(* PLC project Unnamed, Unknown Unnamed 1 *)
(* stored: creationDateTime 2023-03-25T12:40:06, modificationDateTime 2023-03-28T19:18:31 *)

PROGRAM PPXYZ
  VAR
    START AT %IX100.0 : BOOL;
    STOP AT %IX100.1 : BOOL;
    SEN1 AT %IX100.2 : BOOL;
    SEN2 AT %IX100.3 : BOOL;
    CON1 AT %QX100.0 : BOOL;
    CON2 AT %QX100.1 : BOOL;
    GRAP AT %QX100.2 : BOOL;
    X AT %IW100 : INT;
    SPX AT %QW100 : INT;
    SPY AT %QW101 : INT;
    SPZ AT %QW102 : INT;
    DIGRED AT %QW103 : INT;
    VIR1 AT %QX0.0 : BOOL;
    VIR2 AT %QX0.1 : BOOL;
    VIR3 AT %QX0.2 : BOOL;
    VIR4 AT %QX0.3 : BOOL;
    VIR5 AT %QX0.4 : BOOL;
    VIR6 AT %QX0.5 : BOOL;
    VIR7 AT %QX0.6 : BOOL;
    VIR8 AT %QX0.7 : BOOL;
    Block1 AT %QX1.0 : BOOL;
    Block2 AT %QX1.1 : BOOL;
    Block3 AT %QX1.2 : BOOL;
    Block4 AT %QX1.3 : BOOL;
    GRABVIR1 AT %QX2.1 : BOOL;
    GRABVIR2 AT %QX2.2 : BOOL;
    GRABVIR3 AT %QX2.3 : BOOL;
    GRABVIR4 AT %QX2.4 : BOOL;
  END_VAR
  VAR
    TON0 : TON;
    TON1 : TON;
    TON2 : TON;
    TON3 : TON;
    TON4 : TON;
    TON5 : TON;
    TON6 : TON;
    TON7 : TON;
    TON8 : TON;
    TON9 : TON;
    TON10 : TON;
    TON11 : TON;
    TON12 : TON;
    TON13 : TON;
    TON14 : TON;
    TON15 : TON;
    TON16 : TON;
    TON17 : TON;
    TON18 : TON;
    TON19 : TON;
  END_VAR
  VAR  (* added by the conversion: wires and edge detectors of the diagram *)
    _MOVE77_ENO : BOOL;
    _MOVE77_OUT : INT;
    _MOVE8_ENO : BOOL;
    _MOVE8_OUT : INT;
    _MOVE12_ENO : BOOL;
    _MOVE12_OUT : INT;
    _MOVE16_ENO : BOOL;
    _MOVE16_OUT : INT;
    _MOVE20_ENO : BOOL;
    _MOVE20_OUT : INT;
    _MOVE29_ENO : BOOL;
    _MOVE29_OUT : INT;
    _MOVE69_ENO : BOOL;
    _MOVE69_OUT : INT;
    _MOVE40_ENO : BOOL;
    _MOVE40_OUT : INT;
    _MOVE44_ENO : BOOL;
    _MOVE44_OUT : INT;
    _MOVE48_ENO : BOOL;
    _MOVE48_OUT : INT;
    _MOVE52_ENO : BOOL;
    _MOVE52_OUT : INT;
    _MOVE61_ENO : BOOL;
    _MOVE61_OUT : INT;
    _MOVE139_ENO : BOOL;
    _MOVE139_OUT : INT;
    _MOVE186_ENO : BOOL;
    _MOVE186_OUT : INT;
    _MOVE110_ENO : BOOL;
    _MOVE110_OUT : INT;
    _MOVE152_ENO : BOOL;
    _MOVE152_OUT : INT;
    _MOVE114_ENO : BOOL;
    _MOVE114_OUT : INT;
    _MOVE157_ENO : BOOL;
    _MOVE157_OUT : INT;
    _MOVE199_ENO : BOOL;
    _MOVE199_OUT : INT;
    _MOVE161_ENO : BOOL;
    _MOVE161_OUT : INT;
    _MOVE118_ENO : BOOL;
    _MOVE118_OUT : INT;
    _MOVE122_ENO : BOOL;
    _MOVE122_OUT : INT;
    _MOVE165_ENO : BOOL;
    _MOVE165_OUT : INT;
    _MOVE169_ENO : BOOL;
    _MOVE169_OUT : INT;
    _MOVE131_ENO : BOOL;
    _MOVE131_OUT : INT;
    _MOVE178_ENO : BOOL;
    _MOVE178_OUT : INT;
  END_VAR

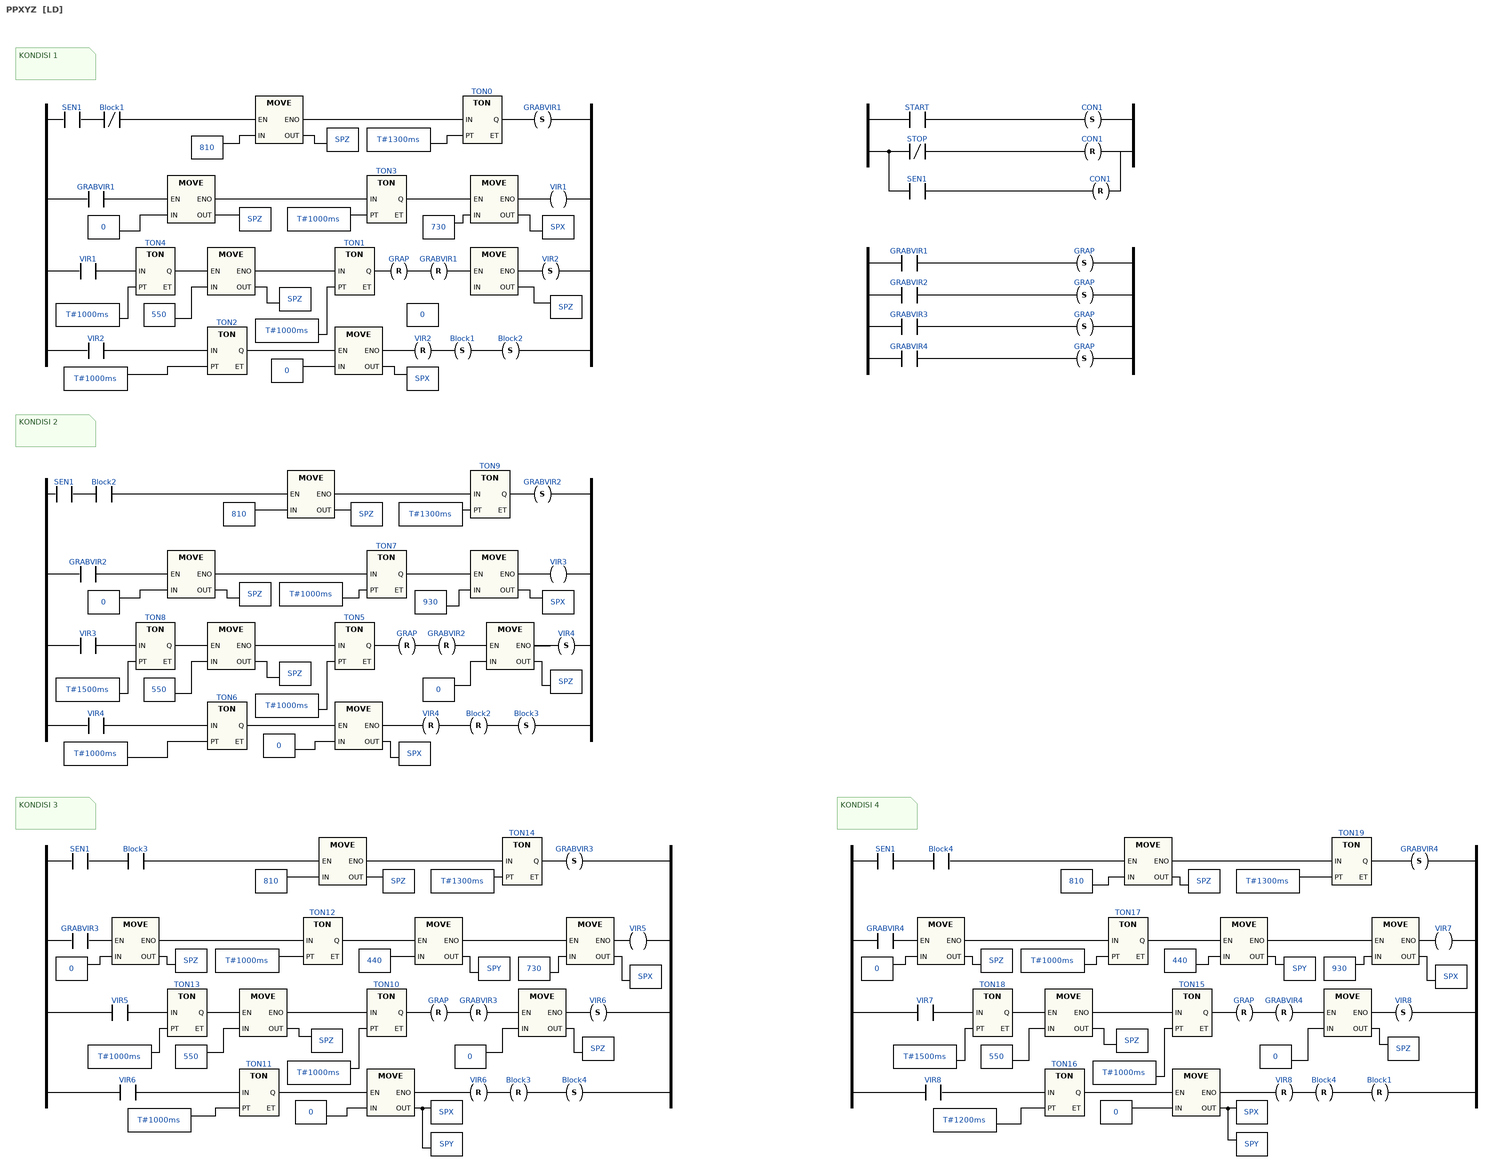
(* LD diagram, written out as Structured Text *)
(* KONDISI 1 *)
_MOVE77_OUT := MOVE(EN := SEN1 AND NOT Block1, IN := 810, ENO => _MOVE77_ENO);
TON0(IN := _MOVE77_ENO, PT := T#1300ms);
IF TON0.Q THEN GRABVIR1 := TRUE; END_IF;
IF START THEN CON1 := TRUE; END_IF;
IF _MOVE77_ENO THEN SPZ := _MOVE77_OUT; END_IF;
IF NOT STOP THEN CON1 := FALSE; END_IF;
IF SEN1 THEN CON1 := FALSE; END_IF;
_MOVE8_OUT := MOVE(EN := GRABVIR1, IN := 0, ENO => _MOVE8_ENO);
TON3(IN := _MOVE8_ENO, PT := T#1000ms);
_MOVE12_OUT := MOVE(EN := TON3.Q, IN := 730, ENO => _MOVE12_ENO);
VIR1 := _MOVE12_ENO;
IF _MOVE8_ENO THEN SPZ := _MOVE8_OUT; END_IF;
IF _MOVE12_ENO THEN SPX := _MOVE12_OUT; END_IF;
IF GRABVIR1 THEN GRAP := TRUE; END_IF;
TON4(IN := VIR1, PT := T#1000ms);
_MOVE16_OUT := MOVE(EN := TON4.Q, IN := 550, ENO => _MOVE16_ENO);
TON1(IN := _MOVE16_ENO, PT := T#1000ms);
IF TON1.Q THEN GRAP := FALSE; END_IF;
IF TON1.Q THEN GRABVIR1 := FALSE; END_IF;
_MOVE20_OUT := MOVE(EN := TON1.Q, ENO => _MOVE20_ENO);
IF _MOVE20_ENO THEN VIR2 := TRUE; END_IF;
IF _MOVE16_ENO THEN SPZ := _MOVE16_OUT; END_IF;
IF GRABVIR2 THEN GRAP := TRUE; END_IF;
IF _MOVE20_ENO THEN SPZ := _MOVE20_OUT; END_IF;
IF GRABVIR3 THEN GRAP := TRUE; END_IF;
TON2(IN := VIR2, PT := T#1000ms);
_MOVE29_OUT := MOVE(EN := TON2.Q, IN := 0, ENO => _MOVE29_ENO);
IF _MOVE29_ENO THEN VIR2 := FALSE; END_IF;
IF _MOVE29_ENO THEN Block1 := TRUE; END_IF;
IF _MOVE29_ENO THEN Block2 := TRUE; END_IF;
IF GRABVIR4 THEN GRAP := TRUE; END_IF;
IF _MOVE29_ENO THEN SPX := _MOVE29_OUT; END_IF;
(* KONDISI 2 *)
_MOVE69_OUT := MOVE(EN := SEN1 AND Block2, IN := 810, ENO => _MOVE69_ENO);
TON9(IN := _MOVE69_ENO, PT := T#1300ms);
IF TON9.Q THEN GRABVIR2 := TRUE; END_IF;
IF _MOVE69_ENO THEN SPZ := _MOVE69_OUT; END_IF;
_MOVE40_OUT := MOVE(EN := GRABVIR2, IN := 0, ENO => _MOVE40_ENO);
TON7(IN := _MOVE40_ENO, PT := T#1000ms);
_MOVE44_OUT := MOVE(EN := TON7.Q, IN := 930, ENO => _MOVE44_ENO);
VIR3 := _MOVE44_ENO;
IF _MOVE40_ENO THEN SPZ := _MOVE40_OUT; END_IF;
IF _MOVE44_ENO THEN SPX := _MOVE44_OUT; END_IF;
TON8(IN := VIR3, PT := T#1500ms);
_MOVE48_OUT := MOVE(EN := TON8.Q, IN := 550, ENO => _MOVE48_ENO);
TON5(IN := _MOVE48_ENO, PT := T#1000ms);
IF TON5.Q THEN GRAP := FALSE; END_IF;
IF TON5.Q THEN GRABVIR2 := FALSE; END_IF;
_MOVE52_OUT := MOVE(EN := TON5.Q, IN := 0, ENO => _MOVE52_ENO);
IF _MOVE52_ENO THEN VIR4 := TRUE; END_IF;
IF _MOVE48_ENO THEN SPZ := _MOVE48_OUT; END_IF;
IF _MOVE52_ENO THEN SPZ := _MOVE52_OUT; END_IF;
TON6(IN := VIR4, PT := T#1000ms);
_MOVE61_OUT := MOVE(EN := TON6.Q, IN := 0, ENO => _MOVE61_ENO);
IF _MOVE61_ENO THEN VIR4 := FALSE; END_IF;
IF _MOVE61_ENO THEN Block2 := FALSE; END_IF;
IF _MOVE61_ENO THEN Block3 := TRUE; END_IF;
IF _MOVE61_ENO THEN SPX := _MOVE61_OUT; END_IF;
(* KONDISI 3 *)
(* KONDISI 4 *)
_MOVE139_OUT := MOVE(EN := SEN1 AND Block3, IN := 810, ENO => _MOVE139_ENO);
TON14(IN := _MOVE139_ENO, PT := T#1300ms);
IF TON14.Q THEN GRABVIR3 := TRUE; END_IF;
_MOVE186_OUT := MOVE(EN := SEN1 AND Block4, IN := 810, ENO => _MOVE186_ENO);
TON19(IN := _MOVE186_ENO, PT := T#1300ms);
IF TON19.Q THEN GRABVIR4 := TRUE; END_IF;
IF _MOVE139_ENO THEN SPZ := _MOVE139_OUT; END_IF;
IF _MOVE186_ENO THEN SPZ := _MOVE186_OUT; END_IF;
_MOVE110_OUT := MOVE(EN := GRABVIR3, IN := 0, ENO => _MOVE110_ENO);
TON12(IN := _MOVE110_ENO, PT := T#1000ms);
_MOVE152_OUT := MOVE(EN := TON12.Q, IN := 440, ENO => _MOVE152_ENO);
_MOVE114_OUT := MOVE(EN := _MOVE152_ENO, IN := 730, ENO => _MOVE114_ENO);
VIR5 := _MOVE114_ENO;
_MOVE157_OUT := MOVE(EN := GRABVIR4, IN := 0, ENO => _MOVE157_ENO);
TON17(IN := _MOVE157_ENO, PT := T#1000ms);
_MOVE199_OUT := MOVE(EN := TON17.Q, IN := 440, ENO => _MOVE199_ENO);
_MOVE161_OUT := MOVE(EN := _MOVE199_ENO, IN := 930, ENO => _MOVE161_ENO);
VIR7 := _MOVE161_ENO;
IF _MOVE110_ENO THEN SPZ := _MOVE110_OUT; END_IF;
IF _MOVE157_ENO THEN SPZ := _MOVE157_OUT; END_IF;
IF _MOVE152_ENO THEN SPY := _MOVE152_OUT; END_IF;
IF _MOVE199_ENO THEN SPY := _MOVE199_OUT; END_IF;
IF _MOVE114_ENO THEN SPX := _MOVE114_OUT; END_IF;
IF _MOVE161_ENO THEN SPX := _MOVE161_OUT; END_IF;
TON13(IN := VIR5, PT := T#1000ms);
_MOVE118_OUT := MOVE(EN := TON13.Q, IN := 550, ENO => _MOVE118_ENO);
TON10(IN := _MOVE118_ENO, PT := T#1000ms);
IF TON10.Q THEN GRAP := FALSE; END_IF;
IF TON10.Q THEN GRABVIR3 := FALSE; END_IF;
_MOVE122_OUT := MOVE(EN := TON10.Q, IN := 0, ENO => _MOVE122_ENO);
IF _MOVE122_ENO THEN VIR6 := TRUE; END_IF;
TON18(IN := VIR7, PT := T#1500ms);
_MOVE165_OUT := MOVE(EN := TON18.Q, IN := 550, ENO => _MOVE165_ENO);
TON15(IN := _MOVE165_ENO, PT := T#1000ms);
IF TON15.Q THEN GRAP := FALSE; END_IF;
IF TON15.Q THEN GRABVIR4 := FALSE; END_IF;
_MOVE169_OUT := MOVE(EN := TON15.Q, IN := 0, ENO => _MOVE169_ENO);
IF _MOVE169_ENO THEN VIR8 := TRUE; END_IF;
IF _MOVE118_ENO THEN SPZ := _MOVE118_OUT; END_IF;
IF _MOVE165_ENO THEN SPZ := _MOVE165_OUT; END_IF;
IF _MOVE122_ENO THEN SPZ := _MOVE122_OUT; END_IF;
IF _MOVE169_ENO THEN SPZ := _MOVE169_OUT; END_IF;
TON11(IN := VIR6, PT := T#1000ms);
_MOVE131_OUT := MOVE(EN := TON11.Q, IN := 0, ENO => _MOVE131_ENO);
IF _MOVE131_ENO THEN VIR6 := FALSE; END_IF;
IF _MOVE131_ENO THEN Block3 := FALSE; END_IF;
IF _MOVE131_ENO THEN Block4 := TRUE; END_IF;
TON16(IN := VIR8, PT := T#1200ms);
_MOVE178_OUT := MOVE(EN := TON16.Q, IN := 0, ENO => _MOVE178_ENO);
IF _MOVE178_ENO THEN VIR8 := FALSE; END_IF;
IF _MOVE178_ENO THEN Block4 := FALSE; END_IF;
IF _MOVE178_ENO THEN Block1 := FALSE; END_IF;
IF _MOVE131_ENO THEN SPX := _MOVE131_OUT; END_IF;
IF _MOVE178_ENO THEN SPX := _MOVE178_OUT; END_IF;
IF _MOVE131_ENO THEN SPY := _MOVE131_OUT; END_IF;
IF _MOVE178_ENO THEN SPY := _MOVE178_OUT; END_IF;
(* drawn but not wired to any output: 0 *)
END_PROGRAM

CONFIGURATION Config0
  RESOURCE Res0 ON PLC
    TASK task0(INTERVAL := T#20ms, PRIORITY := 0);
    PROGRAM instance0 WITH task0 : PPXYZ;
  END_RESOURCE
END_CONFIGURATION
